ABB RobotStudio station: Solution3.rsstn

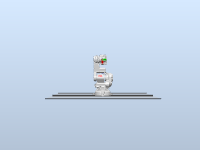
Station Solution3 (saved by RobotStudio 7.0.8683.559)
Controller IRB_140_6kg_0.81m_1
  mechanical unit ROB_1: IRB140_6_81_C_03, 6 joints, base frame (0, 0, 0) mm
Layout (positions relative to the parent item):
  - IRB140_6_81_C_03 [mechanism, from Robots\IRB140_6_81_C_G_03.rslib] at (0, 0, 0) mm; joint values [-0.0132, 0.0296, 0.0033, 0.0093, 0.0241, 0.028] (rad or m)
